  rq_activate_all_grippers(False)
  # end: URCap Program Node
  # begin: URCap Program Node
  #   Source: Robotiq_Grippers, 2.4.0.45103, Robotiq Inc.
  #   Type: Gripper
  $ 17 "Gripper Close (3)" "noBreak"
  if not(gripper_connected[2]):
    popup("Gripper 3 must be connected to run this program.", "No connection", False, True, True)
  end
  if not(rq_is_gripper_activated("3")):
    popup("Gripper 3 is not activated. Go to Installation tab > Gripper to activate it and run the program again.", "Not activated", False, True, True)
  end
  rq_set_pos_spd_for(255, 255, 255, "3")
  rq_wait_pos_spe_for_request(255, 255, 255, "3")
  rq_go_to("3")
  rq_wait("3")
  # end: URCap Program Node
  $ 18 "MoveL" "noBreak"
  $ 19 "Approach_3" "noBreak"
  movel(pose_trans(referencePoin_2, pose_trans(p[-.000149880454, .693597312379, -.374742414510, .017987717953, -2.210197070864, 2.216558983363], Approach_3_p)), a=1.2, v=0.25)
  Pallet_3_sep = False
  if (Pallet_3_cnt >= 1):
    Pallet_3_cnt = 1
  else:
    Pallet_3_cnt = Pallet_3_cnt + 1
  end
  $ 20 "timer_1: Reset"
  timer_1 = 0
  $ 21 "MoveJ"
  $ 22 "Cami_magatz" "breakAfter"
  movej(get_inverse_kin(Cami_magatz_p, qnear=Cami_magatz_q), a=1.3962634015954636, v=1.0471975511965976)
  $ 23 "Pallet_4"
  def Pallet_4_trans(pose):
  return p[pose[0], pose[1], pose[2], 0, 0, 0]
  end
  def Pallet_4_rot(pose):
  return p[0, 0, 0, pose[3], pose[4], pose[5]]
  end
  def Pallet_4_compute_pallet_waypoint(T_base_feature_taught, T_feature_referencePoint_taught, T_referencePoint_approach_taught, T_base_feature, T_base_referencePoint):
  local trans_referencePoint_approach_in_feature_taught = pose_sub(Pallet_4_trans(pose_trans(T_feature_referencePoint_taught, T_referencePoint_approach_taught)), Pallet_4_trans(T_feature_referencePoint_taught))
  local rot_referencePoint_approach_in_feature_taught = pose_trans(Pallet_4_rot(T_feature_referencePoint_taught), pose_trans(Pallet_4_rot(T_referencePoint_approach_taught), pose_inv(Pallet_4_rot(T_feature_referencePoint_taught))))
  T_feature_referencePoint = pose_trans(pose_inv(T_base_feature), T_base_referencePoint)
  rot_referencePoint_approach = pose_trans(pose_inv(Pallet_4_rot(T_feature_referencePoint)), pose_trans(rot_referencePoint_approach_in_feature_taught, Pallet_4_rot(T_feature_referencePoint)))
  T_feature_approach = pose_trans(trans_referencePoint_approach_in_feature_taught, pose_trans(T_feature_referencePoint, rot_referencePoint_approach))
  T_base_approach = pose_trans(T_base_feature, T_feature_approach)
  return T_base_approach
  end
  Pallet_4_tct = 6
  if (Pallet_4_cnt > 6 or Pallet_4_cnt < 1):
    Pallet_4_cnt = 1
  end
  $ 24 "Patterns" "noBreak"
  $ 25 "Grid_Pattern_1" "noBreak"
  $ 30 "Layers" "noBreak"
  if (Pallet_4_cnt < 7):
    Pallet_4_lno = 1
    Pallet_4_lct = Pallet_4_cnt
    global CornerItem_1=pose_trans(p[0.0,0.0,0.0,0.0,0.0,0.0], pose_trans(p[-.000000000000, -.000000000000, -.000000000000, .000000000000, .000000000000, .000000000000], p[.005949599292, -.372700240057, .694671391250, -.017923809946, 2.210134225754, -2.216495424136]))
    global CornerItem_2=pose_trans(p[0.0,0.0,0.0,0.0,0.0,0.0], pose_trans(p[-.000000000000, -.000000000000, -.000000000000, .000000000000, .000000000000, .000000000000], p[.005950540977, -.372700255988, .694671419358, -.017916727829, 2.210126579927, -2.216487728786]))
    global CornerItem_3=pose_trans(p[0.0,0.0,0.0,0.0,0.0,0.0], pose_trans(p[-.000000000000, -.000000000000, -.000000000000, .000000000000, .000000000000, .000000000000], p[.005946645315, -.372700316568, .694671354116, -.017959100293, 2.210169111761, -2.216531106631]))
    global CornerItem_4=pose_trans(p[0.0,0.0,0.0,0.0,0.0,0.0], pose_trans(p[-.000000000000, -.000000000000, -.000000000000, .000000000000, .000000000000, .000000000000], p[.005942968376, -.372700450227, .694671319276, -.017917075683, 2.210174361962, -2.216535908837]))
    Pallet_4_cnt_x = (Pallet_4_lct - 1) % 2
    Pallet_4_cnt_y = floor((Pallet_4_lct - 1) / 2)
    referencePoin_3 = interpolate_pose(interpolate_pose(CornerItem_1, CornerItem_2, Pallet_4_cnt_x/1), interpolate_pose(CornerItem_4, CornerItem_3,Pallet_4_cnt_x/1), Pallet_4_cnt_y/2)
    direction = p[0,0,1,0,0,0]
    referencePoin_3 = pose_add (referencePoin_3,p[0.0*direction[0],0.0*direction[1],0.0*direction[2],0,0,0])
  end
  Approach_4_p = Pallet_4_compute_pallet_waypoint(p[0.0,0.0,0.0,0.0,0.0,0.0], pose_trans(pose_inv(p[0.0,0.0,0.0,0.0,0.0,0.0]), p[0.005949599292351476,-0.3727002400566459,0.6946713912496693,-0.017923809946475345,2.21013422575449,-2.2164954241357937]), p[2.429601367119513E-6,-1.885176733606997E-7,-1.1150026968387294E-7,5.039411101092013E-7,1.6135644595293568E-5,-2.1332892202399765E-5], p[0.0,0.0,0.0,0.0,0.0,0.0], referencePoin_3)
  Approach_4_p = pose_trans(p[0.005949599292351476,-0.3727002400566459,0.6946713912496693,-0.017923809946511392,2.210134225754455,-2.216495424135759], pose_trans(pose_inv(referencePoin_3), Approach_4_p))
  ToolActionPoi_3_p = Pallet_4_compute_pallet_waypoint(p[0.0,0.0,0.0,0.0,0.0,0.0], pose_trans(pose_inv(p[0.0,0.0,0.0,0.0,0.0,0.0]), p[0.005949599292351476,-0.3727002400566459,0.6946713912496693,-0.017923809946475345,2.21013422575449,-2.2164954241357937]), p[0.0,0.0,0.0,0.0,0.0,0.0], p[0.0,0.0,0.0,0.0,0.0,0.0], referencePoin_3)
  ToolActionPoi_3_p = pose_trans(p[0.005949599292351476,-0.3727002400566459,0.6946713912496693,-0.017923809946511392,2.210134225754455,-2.216495424135759], pose_trans(pose_inv(referencePoin_3), ToolActionPoi_3_p))
  Approach_4_p = Pallet_4_compute_pallet_waypoint(p[0.0,0.0,0.0,0.0,0.0,0.0], pose_trans(pose_inv(p[0.0,0.0,0.0,0.0,0.0,0.0]), p[0.005949599292351476,-0.3727002400566459,0.6946713912496693,-0.017923809946475345,2.21013422575449,-2.2164954241357937]), p[2.429601367119513E-6,-1.885176733606997E-7,-1.1150026968387294E-7,5.039411101092013E-7,1.6135644595293568E-5,-2.1332892202399765E-5], p[0.0,0.0,0.0,0.0,0.0,0.0], referencePoin_3)
  Approach_4_p = pose_trans(p[0.005949599292351476,-0.3727002400566459,0.6946713912496693,-0.017923809946511392,2.210134225754455,-2.216495424135759], pose_trans(pose_inv(referencePoin_3), Approach_4_p))
  $ 31 "At Each Item" "noBreak"
  $ 32 "Generated Movements" "noBreak"
  $ 33 "MoveJ" "noBreak"
  $ 34 "Approach_4" "noBreak"
  movej(get_inverse_kin(pose_trans(referencePoin_3, pose_trans(p[-.000106486355, .693597322644, -.374742513164, .017923809946, -2.210134225754, 2.216495424136], Approach_4_p)), qnear=Approach_4_q), a=1.3962634015954636, v=1.0471975511965976)
  $ 35 "MoveL" "noBreak"
  $ 36 "ToolActionPoi_3" "noBreak"
  movel(pose_trans(referencePoin_3, pose_trans(p[-.000106486355, .693597322644, -.374742513164, .017923809946, -2.210134225754, 2.216495424136], ToolActionPoi_3_p)), a=1.2, v=0.25)
  $ 37 "Tool action" "noBreak"
  # begin: URCap Program Node
  #   Source: Robotiq_Grippers, 2.4.0.45103, Robotiq Inc.
  #   Type: Gripper
  $ 38 "Gripper Open (3)" "noBreak"
  if not(gripper_connected[2]):
    popup("Gripper 3 must be connected to run this program.", "No connection", False, True, True)
  end
  if not(rq_is_gripper_activated("3")):
    popup("Gripper 3 is not activated. Go to Installation tab > Gripper to activate it and run the program again.", "Not activated", False, True, True)
  end
  rq_set_pos_spd_for(0, 255, 255, "3")
  rq_wait_pos_spe_for_request(0, 255, 255, "3")
  rq_go_to("3")
  rq_wait("3")
  # end: URCap Program Node
  $ 39 "MoveL" "noBreak"
  $ 40 "Approach_4" "noBreak"
  movel(pose_trans(referencePoin_3, pose_trans(p[-.000106486355, .693597322644, -.374742513164, .017923809946, -2.210134225754, 2.216495424136], Approach_4_p)), a=1.2, v=0.25)
  Pallet_4_sep = False
  if (Pallet_4_cnt >= 6):
    Pallet_4_cnt = 1
  else:
    Pallet_4_cnt = Pallet_4_cnt + 1
  end
  $ 41 "Popup: Peca al magatzem"
  popup("Peca al magatzem", "Message", False, False, blocking=True)
  $ 42 "MoveJ"
  $ 43 "inici" "breakAfter"
  movej(get_inverse_kin(inici_p, qnear=inici_q), a=1.3962634015954636, v=1.0471975511965976)
  end
  end
end
